// TIA Portal V17 export
// export: Created 2025-03-07T09:19:46.6778957Z, ExportSetting WithDefaults, DisplayName Totally Integrated Automation Portal, DisplayVersion V17 Update 8, DisplayName TIA Portal Openness, DisplayVersion V17 Update 8, DisplayName TIA Portal Version Control Interface, DisplayVersion V17, DisplayName SINAMICS Startdrive Advanced, DisplayVersion V17 SP2, DisplayName SINAMICS Startdrive G110M, G120, G120C, G120D, G120P, G115D, DisplayVersion V17 SP2, DisplayName SINAMICS Startdrive G130, G150, S120, S150, SINAMICS MV, S210, DisplayVersion V17 SP2, DisplayName STEP 7 Professional, DisplayVersion V17 Update 8, DisplayName SINUMERIK ONE STEP 7 Toolbox, DisplayVersion V17 Update 12, DisplayName SINUMERIK 840D sl STEP 7 Toolbox, DisplayVersion V17 Update 12, DisplayName STEP 7 Safety, DisplayVersion V17 Update 6, DisplayName WinCC Advanced, DisplayVersion V17 Update 8
TYPE "INCREMENTAL"
// stored: IsFailsafeCompliant false
   STRUCT
      GENERAL_CONDITIONS : Bool;   // CHANGE GENERAL CONDITIONS / GENERAL CONDITIONS
      INITIAL_CONDITIONS : Bool;   // CHANGE INITIAL CONDITIONS / INITIAL CONDITIONS
      ENABLE_REQUEST : Bool;   // ENABLE REQUEST
      DISABLE_REQUEST : Bool;   // DISABLE REQUEST
      "1_MICRA_REQUEST" : Bool;   // 1 MICRA REQUEST
      "10_MICRA_REQUEST" : Bool;   // 10 MICRA REQUEST
      "100_MICRA_REQUEST" : Bool;   // 100 MICRA REQUEST
      "1000_MICRA_REQUEST" : Bool;   // 1000 MICRA REQUEST
      TOGGLE_COMMAND_P : Bool;   // TOGGLE COMAND PULSE / TOGGLE COMMAND PULSE
      TOGGLE_COMMAND : Bool;   // TOGGLE COMMAND AUXILIARY / TOGGLE COMMAND
      GENERAL_CONDITIONS_HELP : Bool;   // GENERAL CONDITIONS HELP
      INITIAL_CONDITIONS_HELP : Bool;   // INITIAL CONDITIONS HELP
      INCREMENTAL_MODE_SELECTED : Bool;   // INCREMENTAL MODE SELECTED
      CONTINIOUS_MODE_SELECTED : Bool;   // CONTINOUS MODE SELECTED / CONTINUOUS MODE SELECTED
      INCREMENTAL_MODES_GENERAL_CONDITIONS : Bool;   // CHANGE GENERAL CONDITIONS / INCREMENTAL MODES GENERAL CONDITIONS
      INCREMENTAL_MODES_INITIAL_CONDITIONS : Bool;   // CHANGE INITIAL CONDITIONS / INCREMENTAL MODES INITIAL CONDITIONS
      "1_MICRA_SELECTED" : Bool;   // 1 MICRA SELECTED
      "10_MICRA_SELECTED" : Bool;   // 10 MICRA SELECTED
      "100_MICRA_SELECTED" : Bool;   // 100 MICRA SELECTED
      "1000_MICRA_SELECTED" : Bool;   // 1000 MICRA SELECTED
      ANY_VALUE_SELECTED : Bool;   // ANY VALUE SELECTED
      "1_MICRA_REQUEST_P" : Bool;   // 1 MICRA REQUEST PULSE
      INCREMENTAL_MODES_GENERAL_CONDITIONS_HELP : Bool;   // INCREMENTAL MODES GENERAL CONDITIONS HELP
      INCREMENTAL_MODES_INITIAL_CONDITIONS_HELP : Bool;   // INCREMENTAL MODES INITIAL CONDITIONS HELP
      WARNING_GONE : Bool;   // WARNING GONE
   END_STRUCT;
END_TYPE
